TYPE (* Reponse sent by the orchestrator *)
  (* Standard: 61499-2; Description: Copyright (c) 2018 fortiss GmbH This program and the accompanying materials are made available under the terms of the Eclipse Public License 2.0 which is available at https://www.eclipse.org/legal/epl-2.0/ SPDX-License-Identifier: EPL-2.0 *)
  (* Version 1.0, 2018-09-26, Jose Cabral, fortiss GmbH *)
  (* ASN.1 tag APPLICATION 1 *)
  OrchestrationForm : STRUCT
    service : ArrowheadService; (* The exact Service that needs to be consumed. This response matches the ServiceRequestForm’s (if that was filled out), but it comes from the exact Service instance with proper metadata and interface identifier (only one). *)
    provider : ArrowheadSystem; (* The Application System description that will provide the Service. *)
    serviceURI : WSTRING; (* The base URL within the Service Provider that will contain the seeked Service. *)
    instruction : WSTRING; (* Optional additional data from the orchestration *)
    authorizationToken : WSTRING; (* The encrypted authorization token. *)
    signature : WSTRING; (* The signature from the Authorization System for the token (verifying the token issuing) *)
    warnings : ARRAY [0..9] OF WSTRING; (* The signature from the Authorization System for the token (verifying the token issuing) *)
  END_STRUCT;
END_TYPE
